FUNCTION_BLOCK AI_D_FF_HYS_TMIN (* Data latch (d) flip flop with a Hysteresis, with a Minimum inter-disposal Time between EO *)
  (* Standard: 61499-1 Annex A; Description: Copyright (c) 2017 fortiss GmbH, HR Agrartechnik GmbH This program and the accompanying materials are made available under the terms of the Eclipse Public License 2.0 which is available at https://www.eclipse.org/legal/epl-2.0/ SPDX-License-Identifier: EPL-2.0 *)
  (* Version 1.0, 2026-05-15, Franz Höpfinger, HR Agrartechnik GmbH, Inital API *)
  PACKAGE adapter::events::unidirectional;
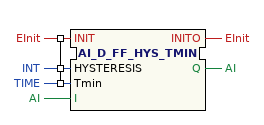
  EVENT_INPUT
    INIT : EInit WITH HYSTERESIS, Tmin; (* Init Request *)
  END_EVENT
  EVENT_OUTPUT
    INITO : EInit; (* Init Confirmation *)
  END_EVENT
  VAR_INPUT
    HYSTERESIS : INT; (* Hysteresis band *)
    Tmin : TIME; (* Minimum inter-arrival time between EI events *)
  END_VAR
  SOCKETS
    I : adapter::types::unidirectional::AI; (* Value to latch *)
  END_SOCKETS
  PLUGS
    Q : adapter::types::unidirectional::AI; (* Latched value *)
  END_PLUGS
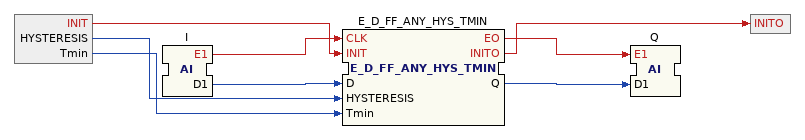
  FBS
    E_D_FF_ANY_HYS_TMIN : logiBUS::signalprocessing::hysteresis::E_D_FF_ANY_HYS_TMIN;
  END_FBS
  EVENT_CONNECTIONS
    I.E1 TO E_D_FF_ANY_HYS_TMIN.CLK;
    E_D_FF_ANY_HYS_TMIN.EO TO Q.E1;
    INIT TO E_D_FF_ANY_HYS_TMIN.INIT;
    E_D_FF_ANY_HYS_TMIN.INITO TO INITO;
  END_CONNECTIONS
  DATA_CONNECTIONS
    I.D1 TO E_D_FF_ANY_HYS_TMIN.D;
    E_D_FF_ANY_HYS_TMIN.Q TO Q.D1;
    HYSTERESIS TO E_D_FF_ANY_HYS_TMIN.HYSTERESIS;
    Tmin TO E_D_FF_ANY_HYS_TMIN.Tmin;
  END_CONNECTIONS
END_FUNCTION_BLOCK
